LIN {X 0,Y 67.892,Z 663.193,A -85,B 0,C 180,E1 -30054.056,E2 -30054.056} C_VEL
LIN {X 0,Y 67.877,Z 661.678,A -85,B 0,C 180,E1 -30057.03,E2 -30057.03} C_VEL
LIN {X 0,Y 67.591,Z 659.063,A -85,B 0,C 180,E1 -30065.966,E2 -30065.966} C_VEL
LIN {X 0,Y 66.795,Z 659.556,A -85,B 0,C 180,E1 -30072.145,E2 -30072.145} C_VEL
LIN {X 0,Y 66.253,Z 660.862,A -85,B 0,C 180,E1 -30078.554,E2 -30078.554} C_VEL
LIN {X 0,Y 66.081,Z 663.554,A -85,B 0,C 180,E1 -30087.771,E2 -30087.771} C_VEL
LIN {X 0,Y 65.88,Z 666.752,A -85,B 0,C 180,E1 -30094.742,E2 -30094.742} C_VEL
LIN {X 0,Y 65.314,Z 670.634,A -85,B 0,C 180,E1 -30101.122,E2 -30101.122} C_VEL
LIN {X 0,Y 65.053,Z 672.114,A -85,B 0,C 180,E1 -30103.403,E2 -30103.403} C_VEL
LIN {X 0,Y 64.242,Z 674.05,A -85,B 0,C 180,E1 -30105.561,E2 -30105.561} C_VEL
LIN {X 0,Y 56.97,Z 682.772,A -85,B 0,C 180,E1 -30111.908,E2 -30111.908} C_VEL
LIN {X 0,Y 49.93,Z 690.356,A -85,B 0,C 180,E1 -30120.477,E2 -30120.477} C_VEL
LIN {X 0,Y 44.172,Z 696.48,A -85,B 0,C 180,E1 -30131.437,E2 -30131.437} C_VEL
LIN {X 0,Y 40.125,Z 701.384,A -85,B 0,C 180,E1 -30144.967,E2 -30144.967} C_VEL
LIN {X 0,Y 38.519,Z 705.175,A -85,B 0,C 180,E1 -30160.503,E2 -30160.503} C_VEL
LIN {X 0,Y 40.41,Z 708.443,A -85,B 0,C 180,E1 -30179.597,E2 -30179.597} C_VEL
LIN {X 0,Y 40.756,Z 708.641,A -85,B 0,C 180,E1 -30181.142,E2 -30181.142} C_VEL
LIN {X 0,Y 42.353,Z 709.992,A -85,B 0,C 180,E1 -30191.574,E2 -30191.574} C_VEL
LIN {X 0,Y 37.093,Z 714.089,A -85,B 0,C 180,E1 -30229.083,E2 -30229.083} C_VEL
LIN {X 0,Y 39.796,Z 715.634,A -85,B 0,C 180,E1 -30245.07,E2 -30245.07} C_VEL
LIN {X 0,Y 40.189,Z 716.922,A -85,B 0,C 180,E1 -30247.22,E2 -30247.22} C_VEL
LIN {X 0,Y 40.574,Z 719.147,A -85,B 0,C 180,E1 -30251.84,E2 -30251.84} C_VEL
LIN {X 0,Y 40.438,Z 721.815,A -85,B 0,C 180,E1 -30260.585,E2 -30260.585} C_VEL
LIN {X 0,Y 41.271,Z 724.287,A -85,B 0,C 180,E1 -30269.389,E2 -30269.389} C_VEL
LIN {X 0,Y 42.926,Z 726.222,A -85,B 0,C 180,E1 -30273.606,E2 -30273.606} C_VEL
LIN {X 0,Y 45.902,Z 728.976,A -85,B 0,C 180,E1 -30277.77,E2 -30277.77} C_VEL
LIN {X 0,Y 45.942,Z 729.1,A -85,B 0,C 180,E1 -30280.118,E2 -30280.118} C_VEL
LIN {X 0,Y 39.342,Z 722.138,A -85,B 0,C 180,E1 -30297.605,E2 -30297.605} C_VEL
LIN {X 0,Y 38.06,Z 719.237,A -85,B 0,C 180,E1 -30305.461,E2 -30305.461} C_VEL
LIN {X 0,Y 37.438,Z 719.028,A -85,B 0,C 180,E1 -30307.959,E2 -30307.959} C_VEL
LIN {X 0,Y 34.428,Z 717.685,A -85,B 0,C 180,E1 -30318.232,E2 -30318.232} C_VEL
LIN {X 0,Y 31.542,Z 714.719,A -85,B 0,C 180,E1 -30336.408,E2 -30336.408} C_VEL
LIN {X 0,Y 32.173,Z 710.675,A -85,B 0,C 180,E1 -30355.918,E2 -30355.918} C_VEL
LIN {X 0,Y 36.173,Z 705.457,A -85,B 0,C 180,E1 -30372.857,E2 -30372.857} C_VEL
LIN {X 0,Y 41.849,Z 698.611,A -85,B 0,C 180,E1 -30387.122,E2 -30387.122} C_VEL
LIN {X 0,Y 49.307,Z 689.952,A -85,B 0,C 180,E1 -30397.912,E2 -30397.912} C_VEL
LIN {X 0,Y 56.205,Z 681.277,A -85,B 0,C 180,E1 -30404.797,E2 -30404.797} C_VEL
LIN {X 0,Y 61.975,Z 673.087,A -85,B 0,C 180,E1 -30409.462,E2 -30409.462} C_VEL
LIN {X 0,Y 62.888,Z 669.955,A -85,B 0,C 180,E1 -30413.581,E2 -30413.581} C_VEL
LIN {X 0,Y 63.386,Z 668.05,A -85,B 0,C 180,E1 -30416.357,E2 -30416.357} C_VEL
LIN {X 0,Y 63.463,Z 666.54,A -85,B 0,C 180,E1 -30419.997,E2 -30419.997} C_VEL
LIN {X 0,Y 63.4,Z 664.968,A -85,B 0,C 180,E1 -30426.362,E2 -30426.362} C_VEL
LIN {X 0,Y 62.478,Z 665.594,A -85,B 0,C 180,E1 -30432.999,E2 -30432.999} C_VEL
LIN {X 0,Y 61.571,Z 667.998,A -85,B 0,C 180,E1 -30444.04,E2 -30444.04} C_VEL
LIN {X 0,Y 61.005,Z 670.74,A -85,B 0,C 180,E1 -30451.424,E2 -30451.424} C_VEL
LIN {X 0,Y 60.484,Z 672.812,A -85,B 0,C 180,E1 -30455.563,E2 -30455.563} C_VEL
LIN {X 0,Y 59.946,Z 674.722,A -85,B 0,C 180,E1 -30459.055,E2 -30459.055} C_VEL
LIN {X 0,Y 59.175,Z 676.212,A -85,B 0,C 180,E1 -30460.913,E2 -30460.913} C_VEL
LIN {X 0,Y 51.584,Z 684.492,A -85,B 0,C 180,E1 -30467.052,E2 -30467.052} C_VEL
LIN {X 0,Y 43.88,Z 691.962,A -85,B 0,C 180,E1 -30475.895,E2 -30475.895} C_VEL
LIN {X 0,Y 37.479,Z 697.979,A -85,B 0,C 180,E1 -30487.963,E2 -30487.963} C_VEL
LIN {X 0,Y 32.987,Z 702.79,A -85,B 0,C 180,E1 -30503.874,E2 -30503.874} C_VEL
LIN {X 0,Y 31.474,Z 706.491,A -85,B 0,C 180,E1 -30522.891,E2 -30522.891} C_VEL
LIN {X 0,Y 33.87,Z 709.448,A -85,B 0,C 180,E1 -30543.909,E2 -30543.909} C_VEL
LIN {X 0,Y 34.358,Z 709.915,A -85,B 0,C 180,E1 -30547.841,E2 -30547.841} C_VEL
LIN {X 0,Y 32.111,Z 711.301,A -85,B 0,C 180,E1 -30558.966,E2 -30558.966} C_VEL
LIN {X 0,Y 29.842,Z 713.885,A -85,B 0,C 180,E1 -30586.384,E2 -30586.384} C_VEL
LIN {X 0,Y 35.873,Z 716.823,A -85,B 0,C 180,E1 -30617.462,E2 -30617.462} C_VEL
LIN {X 0,Y 42.926,Z 726.222,A -85,B 0,C 180,E1 -30633.606,E2 -30633.606} C_VEL
LIN {X 0,Y 43.226,Z 726.666,A -85,B 0,C 180,E1 -30635.275,E2 -30635.275} C_VEL
LIN {X 0,Y 42.579,Z 726.296,A -85,B 0,C 180,E1 -30638.485,E2 -30638.485} C_VEL
LIN {X 0,Y 40.755,Z 724.776,A -85,B 0,C 180,E1 -30642.459,E2 -30642.459} C_VEL
LIN {X 0,Y 34.737,Z 719.612,A -85,B 0,C 180,E1 -30651.988,E2 -30651.988} C_VEL
LIN {X 0,Y 32.378,Z 718.273,A -85,B 0,C 180,E1 -30657.734,E2 -30657.734} C_VEL
LIN {X 0,Y 31.974,Z 718.117,A -85,B 0,C 180,E1 -30659.081,E2 -30659.081} C_VEL
LIN {X 0,Y 30.977,Z 717.87,A -85,B 0,C 180,E1 -30663.028,E2 -30663.028} C_VEL
LIN {X 0,Y 27.407,Z 716.478,A -85,B 0,C 180,E1 -30675.156,E2 -30675.156} C_VEL
LIN {X 0,Y 24.38,Z 713.426,A -85,B 0,C 180,E1 -30698.302,E2 -30698.302} C_VEL
LIN {X 0,Y 25.854,Z 709.289,A -85,B 0,C 180,E1 -30722.951,E2 -30722.951} C_VEL
LIN {X 0,Y 29.133,Z 705.888,A -85,B 0,C 180,E1 -30736.38,E2 -30736.38} C_VEL
LIN {X 0,Y 34.429,Z 700.616,A -85,B 0,C 180,E1 -30750.197,E2 -30750.197} C_VEL
LIN {X 0,Y 42.914,Z 692.284,A -85,B 0,C 180,E1 -30762.546,E2 -30762.546} C_VEL
LIN {X 0,Y 51.387,Z 683.129,A -85,B 0,C 180,E1 -30770.317,E2 -30770.317} C_VEL
LIN {X 0,Y 56.546,Z 676.835,A -85,B 0,C 180,E1 -30773.943,E2 -30773.943} C_VEL
LIN {X 0,Y 57.704,Z 675.167,A -85,B 0,C 180,E1 -30775.111,E2 -30775.111} C_VEL
LIN {X 0,Y 58.502,Z 673.255,A -85,B 0,C 180,E1 -30778.104,E2 -30778.104} C_VEL
LIN {X 0,Y 58.792,Z 672.308,A -85,B 0,C 180,E1 -30779.997,E2 -30779.997} C_VEL
LIN {X 0,Y 58.862,Z 670.663,A -85,B 0,C 180,E1 -30786.855,E2 -30786.855} C_VEL
LIN {X 0,Y 57.723,Z 671.488,A -85,B 0,C 180,E1 -30794.091,E2 -30794.091} C_VEL
LIN {X 0,Y 56.916,Z 672.903,A -85,B 0,C 180,E1 -30801.74,E2 -30801.74} C_VEL
LIN {X 0,Y 56.075,Z 675.086,A -85,B 0,C 180,E1 -30808.666,E2 -30808.666} C_VEL
LIN {X 0,Y 55.084,Z 677.464,A -85,B 0,C 180,E1 -30814.05,E2 -30814.05} C_VEL
LIN {X 0,Y 54.12,Z 678.816,A -85,B 0,C 180,E1 -30815.778,E2 -30815.778} C_VEL
LIN {X 0,Y 45.188,Z 687.579,A -85,B 0,C 180,E1 -30822.362,E2 -30822.362} C_VEL
LIN {X 0,Y 36.878,Z 694.635,A -85,B 0,C 180,E1 -30831.718,E2 -30831.718} C_VEL
LIN {X 0,Y 30.955,Z 699.475,A -85,B 0,C 180,E1 -30842.981,E2 -30842.981} C_VEL
LIN {X 0,Y 25.855,Z 704.176,A -85,B 0,C 180,E1 -30862.174,E2 -30862.174} C_VEL
LIN {X 0,Y 24.516,Z 707.786,A -85,B 0,C 180,E1 -30886.643,E2 -30886.643} C_VEL
LIN {X 0,Y 26.112,Z 709.602,A -85,B 0,C 180,E1 -30902.551,E2 -30902.551} C_VEL
LIN {X 0,Y 26.619,Z 710.174,A -85,B 0,C 180,E1 -30907.632,E2 -30907.632} C_VEL
LIN {X 0,Y 23.777,Z 711.792,A -85,B 0,C 180,E1 -30923.768,E2 -30923.768} C_VEL
LIN {X 0,Y 23.731,Z 714.58,A -85,B 0,C 180,E1 -30960.007,E2 -30960.007} C_VEL
LIN {X 0,Y 33.88,Z 717.845,A -85,B 0,C 180,E1 -30992.137,E2 -30992.137} C_VEL
LIN {X 0,Y 37.787,Z 722.054,A -85,B 0,C 180,E1 -30999.106,E2 -30999.106} C_VEL
LIN {X 0,Y 37.827,Z 722.128,A -85,B 0,C 180,E1 -31002.013,E2 -31002.013} C_VEL
LIN {X 0,Y 34.574,Z 718.639,A -85,B 0,C 180,E1 -31011.513,E2 -31011.513} C_VEL
LIN {X 0,Y 31.974,Z 718.117,A -85,B 0,C 180,E1 -31019.081,E2 -31019.081} C_VEL
LIN {X 0,Y 29.949,Z 717.592,A -85,B 0,C 180,E1 -31025.116,E2 -31025.116} C_VEL
LIN {X 0,Y 27.548,Z 716.786,A -85,B 0,C 180,E1 -31031.049,E2 -31031.049} C_VEL
LIN {X 0,Y 22.471,Z 714.729,A -85,B 0,C 180,E1 -31044.366,E2 -31044.366} C_VEL
LIN {X 0,Y 18.588,Z 712.107,A -85,B 0,C 180,E1 -31063.487,E2 -31063.487} C_VEL
LIN {X 0,Y 18.264,Z 709.888,A -85,B 0,C 180,E1 -31081.24,E2 -31081.24} C_VEL
LIN {X 0,Y 18.849,Z 709.089,A -85,B 0,C 180,E1 -31086.763,E2 -31086.763} C_VEL
LIN {X 0,Y 24.615,Z 704.354,A -85,B 0,C 180,E1 -31108.962,E2 -31108.962} C_VEL
LIN {X 0,Y 32.861,Z 697.72,A -85,B 0,C 180,E1 -31124.285,E2 -31124.285} C_VEL
LIN {X 0,Y 42.435,Z 689.405,A -85,B 0,C 180,E1 -31133.641,E2 -31133.641} C_VEL
LIN {X 0,Y 51.369,Z 680.323,A -85,B 0,C 180,E1 -31139.349,E2 -31139.349} C_VEL
LIN {X 0,Y 52.494,Z 679.049,A -85,B 0,C 180,E1 -31139.997,E2 -31139.997} C_VEL
LIN {X 0,Y 53.859,Z 677.253,A -85,B 0,C 180,E1 -31141.866,E2 -31141.866} C_VEL
LIN {X 0,Y 53.952,Z 676.16,A -85,B 0,C 180,E1 -31147.482,E2 -31147.482} C_VEL
LIN {X 0,Y 52.111,Z 677.701,A -85,B 0,C 180,E1 -31159.236,E2 -31159.236} C_VEL
LIN {X 0,Y 51.356,Z 678.932,A -85,B 0,C 180,E1 -31164.236,E2 -31164.236} C_VEL
LIN {X 0,Y 50.457,Z 680.412,A -85,B 0,C 180,E1 -31168.534,E2 -31168.534} C_VEL
LIN {X 0,Y 48.71,Z 682.222,A -85,B 0,C 180,E1 -31170.023,E2 -31170.023} C_VEL
LIN {X 0,Y 39.173,Z 690.495,A -85,B 0,C 180,E1 -31176.147,E2 -31176.147} C_VEL
LIN {X 0,Y 30.164,Z 697.206,A -85,B 0,C 180,E1 -31185.638,E2 -31185.638} C_VEL
LIN {X 0,Y 22.429,Z 702.593,A -85,B 0,C 180,E1 -31201.946,E2 -31201.946} C_VEL
LIN {X 0,Y 17.745,Z 706.832,A -85,B 0,C 180,E1 -31229.979,E2 -31229.979} C_VEL
LIN {X 0,Y 17.737,Z 709.051,A -85,B 0,C 180,E1 -31253.32,E2 -31253.32} C_VEL
LIN {X 0,Y 18.191,Z 710.48,A -85,B 0,C 180,E1 -31269.418,E2 -31269.418} C_VEL
LIN {X 0,Y 16.344,Z 713.686,A -85,B 0,C 180,E1 -31320.01,E2 -31320.01} C_VEL
LIN {X 0,Y 27.173,Z 717.031,A -85,B 0,C 180,E1 -31359.134,E2 -31359.134} C_VEL
LIN {X 0,Y 29.111,Z 717.494,A -85,B 0,C 180,E1 -31363.611,E2 -31363.611} C_VEL
LIN {X 0,Y 24.853,Z 716.708,A -85,B 0,C 180,E1 -31375.577,E2 -31375.577} C_VEL
LIN {X 0,Y 20.512,Z 715.258,A -85,B 0,C 180,E1 -31389.983,E2 -31389.983} C_VEL
LIN {X 0,Y 17.249,Z 712.117,A -85,B 0,C 180,E1 -31421.777,E2 -31421.777} C_VEL
LIN {X 0,Y 18.849,Z 709.089,A -85,B 0,C 180,E1 -31446.763,E2 -31446.763} C_VEL
LIN {X 0,Y 20.948,Z 706.678,A -85,B 0,C 180,E1 -31461.085,E2 -31461.085} C_VEL
LIN {X 0,Y 23.136,Z 704.053,A -85,B 0,C 180,E1 -31473.816,E2 -31473.816} C_VEL
LIN {X 0,Y 30.374,Z 697.179,A -85,B 0,C 180,E1 -31495.264,E2 -31495.264} C_VEL
LIN {X 0,Y 34.613,Z 693.806,A -85,B 0,C 180,E1 -31499.789,E2 -31499.789} C_VEL
LIN {X 0,Y 44.039,Z 685.924,A -85,B 0,C 180,E1 -31504.871,E2 -31504.871} C_VEL
LIN {X 0,Y 48.662,Z 681.527,A -85,B 0,C 180,E1 -31506.818,E2 -31506.818} C_VEL
LIN {X 0,Y 48.561,Z 681.448,A -85,B 0,C 180,E1 -31508.318,E2 -31508.318} C_VEL
LIN {X 0,Y 47.05,Z 682.482,A -85,B 0,C 180,E1 -31517.379,E2 -31517.379} C_VEL
LIN {X 0,Y 45.58,Z 683.974,A -85,B 0,C 180,E1 -31522.291,E2 -31522.291} C_VEL
LIN {X 0,Y 35.447,Z 692.128,A -85,B 0,C 180,E1 -31526.825,E2 -31526.825} C_VEL
LIN {X 0,Y 25.561,Z 698.729,A -85,B 0,C 180,E1 -31534.401,E2 -31534.401} C_VEL
LIN {X 0,Y 16.438,Z 704.012,A -85,B 0,C 180,E1 -31550.08,E2 -31550.08} C_VEL
LIN {X 0,Y 10.58,Z 708.15,A -85,B 0,C 180,E1 -31589.965,E2 -31589.965} C_VEL
LIN {X 0,Y 10.409,Z 709.221,A -85,B 0,C 180,E1 -31608.551,E2 -31608.551} C_VEL
LIN {X 0,Y 9.659,Z 710.578,A -85,B 0,C 180,E1 -31633.339,E2 -31633.339} C_VEL
LIN {X 0,Y 15.133,Z 714.506,A -85,B 0,C 180,E1 -31719.09,E2 -31719.09} C_VEL
LIN {X 0,Y 17.184,Z 715.028,A -85,B 0,C 180,E1 -31723.914,E2 -31723.914} C_VEL
LIN {X 0,Y 16.712,Z 714.869,A -85,B 0,C 180,E1 -31729.904,E2 -31729.904} C_VEL
LIN {X 0,Y 10.473,Z 711.958,A -85,B 0,C 180,E1 -31770.035,E2 -31770.035} C_VEL
LIN {X 0,Y 13.251,Z 708.002,A -85,B 0,C 180,E1 -31822.756,E2 -31822.756} C_VEL
LIN {X 0,Y 20.041,Z 703.904,A -85,B 0,C 180,E1 -31842.921,E2 -31842.921} C_VEL
LIN {X 0,Y 29.941,Z 697.266,A -85,B 0,C 180,E1 -31856.21,E2 -31856.21} C_VEL
LIN {X 0,Y 34.613,Z 693.806,A -85,B 0,C 180,E1 -31859.789,E2 -31859.789} C_VEL
LIN {X 0,Y 34.518,Z 693.69,A -85,B 0,C 180,E1 -31861.162,E2 -31861.162} C_VEL
LIN {X 0,Y 32.898,Z 694.491,A -85,B 0,C 180,E1 -31863.811,E2 -31863.811} C_VEL
LIN {X 0,Y 28.948,Z 696.743,A -85,B 0,C 180,E1 -31867.596,E2 -31867.596} C_VEL
LIN {X 0,Y 22.792,Z 700.129,A -85,B 0,C 180,E1 -31872.283,E2 -31872.283} C_VEL
LIN {X 0,Y 17.997,Z 702.57,A -85,B 0,C 180,E1 -31877.167,E2 -31877.167} C_VEL
LIN {X 0,Y 10.758,Z 705.941,A -85,B 0,C 180,E1 -31888.421,E2 -31888.421} C_VEL
LIN {X 0,Y 8.334,Z 706.952,A -85,B 0,C 180,E1 -31894.522,E2 -31894.522} C_VEL
LIN {X 0,Y 3.386,Z 709.45,A -85,B 0,C 180,E1 -31949.89,E2 -31949.89} C_VEL
LIN {X 0,Y 2.678,Z 710.965,A -85,B 0,C 180,E1 -32077.091,E2 -32077.091} C_VEL
LIN {X 0,Y 3.653,Z 711,A -85,B 0,C 180,E1 -32113.054,E2 -32113.054} C_VEL
LIN {X 0,Y 10.462,Z 706.648,A -85,B 0,C 180,E1 -32215.652,E2 -32215.652} C_VEL
LIN {X 0,Y 17.578,Z 703.258,A -85,B 0,C 180,E1 -32223.443,E2 -32223.443} C_VEL
LIN {X 0,Y 28.55,Z 696.811,A -85,B 0,C 180,E1 -32229.975,E2 -32229.975} C_VEL
LIN {X 0,Y 35.984,Z 691.641,A -85,B 0,C 180,E1 -32232.386,E2 -32232.386} C_VEL
LIN {X 0,Y 36.368,Z 691.267,A -85,B 0,C 180,E1 -32234.896,E2 -32234.896} C_VEL
LIN {X 0,Y 25.818,Z 698.204,A -85,B 0,C 180,E1 -32237.64,E2 -32237.64} C_VEL
LIN {X 0,Y 15.33,Z 703.787,A -85,B 0,C 180,E1 -32243.462,E2 -32243.462} C_VEL
LIN {X 0,Y 8.334,Z 706.952,A -85,B 0,C 180,E1 -32254.522,E2 -32254.522} C_VEL
LIN {X 0,Y 8.334,Z 706.952,A -85,B 0,C 180,E1 -32254.522,E2 -32254.522}

QRS_NEXT_CUT()

QRS_NEXT()
QRS_HOME()

END
